{attribute 'GeneratedUsingTerminal: '}
{attribute addProperty BoxType ""}
{attribute addProperty Id "_defaultAT %I*SyncUnitTasks_1988CF1B36"}
{attribute addProperty CRC "328675477"}
{attribute addProperty Size "36"}
TYPE SyncUnits_13973095 :
STRUCT
	{attribute addProperty Name "_default"}
	_default : SyncUnitTasks_1988CF1B;
END_STRUCT
END_TYPE

(* stored: Version 1.2.0.0, ProductVersion 3.1.4024.9
   DUT SyncUnits_13973095: Id {b8539510-9860-02a0-0166-6c100a46ba74} *)
